// ---- GlobalTextList.TcGTLO
TEXTLIST GlobalTextList
  117 = ' MUST BE DISABLED'
  118 = ' MUST BE DISABLED TO RESUME'
  119 = ' MUST BE DISABLED TO RESUME NORMAL OPERATIONS'
  135 = ' MUST BE ENABLED FOR THRESHOLD AND FORCED CHECKS'
  134 = ' WILL PERFORM CHECK OPERATION ONCE AS NEXT TASK'
  33 = '%d'
  29 = '%i'
  55 = '%s'
  96 = '+1'
  126 = '+10'
  98 = '-1'
  127 = '-10'
  128 = '-50'
  4 = '1'
  5 = '2'
  70 = 'Auto Load'
  69 = 'Auto Unload'
  68 = 'AutoUnload'
  31 = 'Average Part Time'
  28 = 'Average Part Time: %d'
  165 = 'Backlash'
  64 = 'Batch'
  61 = 'Batch Process'
  170 = 'Box and Circle'
  24 = 'Clear Output'
  13 = 'Complete'
  35 = 'Completed'
  58 = 'Completed Part Count'
  18 = 'Completed Parts'
  41 = 'Completed Parts (Last 10)'
  75 = 'Completed Parts (newest first)'
  57 = 'CompletedPart Count'
  62 = 'Continual Process'
  1 = 'Create Part'
  111 = 'Diagnostics'
  110 = 'Enable / Disable'
  109 = 'Enable / Disable Position Check'
  121 = 'Enable / Disabling Position Checking'
  108 = 'Enable Position Check'
  122 = 'Enabling / Disabling Position Checking'
  164 = 'Encoder Slip'
  80 = 'End Effector'
  82 = 'End Effector 1'
  84 = 'End Effector Closed'
  86 = 'End Effector Grasp'
  83 = 'End Effector Open'
  85 = 'End Effector Part'
  107 = 'Error'
  157 = 'Fingers \nClosed'
  156 = 'Fingers \nOpen'
  90 = 'Fingers Closed'
  89 = 'Fingers Open'
  160 = 'Fixture'
  151 = 'Fofrces'
  154 = 'Force and Torqu Sensor'
  115 = 'Force Check'
  132 = 'Force Check Next'
  152 = 'Forces'
  136 = 'FT Sensor Controls'
  144 = 'Fx'
  143 = 'Fx (N)'
  145 = 'Fy'
  146 = 'Fz'
  159 = 'Grasped \nPart'
  158 = 'Grasped Part'
  155 = 'Gripper\nBody'
  91 = 'Gripper Body'
  21 = 'I1'
  92 = 'Induced Joint Error'
  99 = 'Induced Joint Error  (In 1/100 rad)'
  169 = 'Induced Robot Joint Error  (In 1/10 degrees)'
  105 = 'Induced Robot Joint Error  (In 1/100 rad)'
  39 = 'Input Position'
  3 = 'Insert Part'
  97 = 'J1'
  100 = 'J2'
  101 = 'J3'
  102 = 'J4'
  103 = 'J5'
  104 = 'J6'
  106 = 'Joint'
  23 = 'Load Input'
  166 = 'Mode'
  116 = 'MUST BE DISABLED'
  120 = 'MUST BE ENABLED FOR THRESHOLD AND FORCED CHECKS'
  147 = 'Newton-meter (N-m)'
  141 = 'Newtons'
  142 = 'Newtons (N)'
  171 = 'NIST Logo'
  22 = 'O1'
  163 = 'Off'
  63 = 'On Demand'
  131 = 'ONE TIME OPERATION'
  44 = 'Online Time'
  40 = 'Output Position'
  114 = 'Part Between Checks'
  124 = 'Part Between Checks Threshold'
  112 = 'Part Between Pos'
  32 = 'Part Count'
  30 = 'Part Count %i'
  27 = 'Part Count: %i'
  140 = 'Part Data Controls'
  8 = 'Part Fixture Time: '
  9 = 'Part Fixture Time: %s'
  88 = 'Part Grasped'
  59 = 'Part Number'
  15 = 'Part Removed'
  12 = 'Part Time: %d'
  11 = 'Part Time: %i'
  10 = 'Part Time: %s'
  36 = 'Part Type'
  113 = 'Parts Since Last Check'
  76 = 'Parts Since Pos Check'
  54 = 'Pick Frame'
  17 = 'Pick From WF'
  53 = 'Pick Location'
  60 = 'Place Frame'
  14 = 'Placed In WF'
  93 = 'Position Check'
  129 = 'Position Check Assigned Next'
  77 = 'Position Check Diagnostics'
  66 = 'Process Mode:\n%s'
  25 = 'Process Status:'
  26 = 'Process Status:\n%s'
  67 = 'Process Type:\n%s'
  51 = 'p_tas'
  2 = 'Remove Part'
  172 = 'Reserved'
  79 = 'Robot'
  78 = 'Robot Data Controls'
  130 = 'Sensor State'
  125 = 'Set at 50'
  123 = 'Settings'
  42 = 'Status'
  47 = 'Status\n%s'
  43 = 'Status: '
  137 = 'Switch FT Sensor Data Monitoring'
  138 = 'Switch FT Sensor Data Recording'
  139 = 'Switch Part Data Recording'
  65 = 'Switch Process Type'
  71 = 'Switch TCP/IP Data'
  72 = 'Switch TCP/IP Data Collection'
  74 = 'Switch TCP/IP Data Monitoring'
  73 = 'Switch TCP/IP Data Recording'
  94 = 'System Process'
  95 = 'System Settings'
  50 = 'Task'
  48 = 'Task Status\n%s'
  153 = 'Torques'
  34 = 'Trans'
  56 = 'Transfer'
  148 = 'Tx'
  149 = 'Ty'
  150 = 'Tz'
  19 = 'UR3'
  167 = 'UR3 Mode'
  46 = 'UR3 Power'
  45 = 'UR3 Status'
  173 = 'UR3 Task'
  20 = 'UR5'
  161 = 'UR5 Kinematic Chain'
  162 = 'UR5 Kinematic Chain Testing'
  168 = 'UR5 Mode'
  52 = 'UR5 Power'
  6 = 'WF1'
  7 = 'WF2'
  133 = 'WILL PERFORM CHECK OPERATION ONCE AS NEXT TASK'
  87 = 'Work Fix'
  16 = 'Work Fixture'
  81 = 'Work Fixtures'
  38 = 'Workfixture'
  37 = 'Workfixture Time (s)'
  0 = 'Workfixtures'
  49 = 'Workframe'
END_TEXTLIST

// ---- VISUs/ForceAndTorque.TcVIS
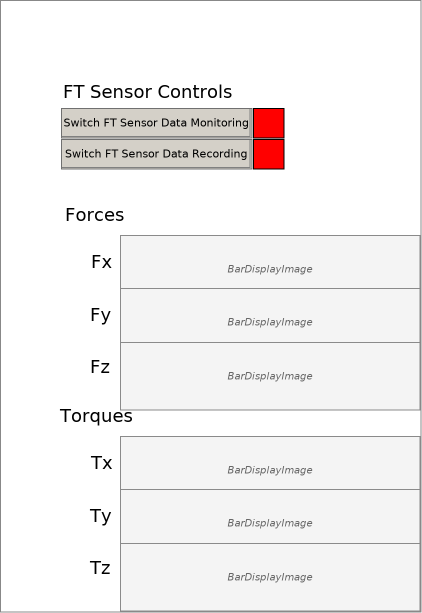
VISUALIZATION ForceAndTorque  // 422x613
    BarDisplayImage (120,235 300x68), value: Global.stFTData.Fx/10000, style: BarDisplayImage-Gray, scale format: %.1f, scale -5..5
        p518627256: Newtons (N)
    BarDisplayImage (120,288 300x68), value: Global.stFTData.Fy/10000, style: BarDisplayImage-Gray, scale format: %.1f, scale -5..5
        p518627256: Newtons (N)
    BarDisplayImage (120,342 300x68), value: Global.stFTData.Fz/10000, style: BarDisplayImage-Gray, scale format: %.1f, scale -5..5
        p518627256: Newtons (N)
    Label (88,247 34x30), "Fx"
    Label (87,300 34x30), "Fy"
    Label (87,352 34x30), "Fz"
    BarDisplayImage (120,436 300x68), value: Global.stFTData.Tx/100000, style: BarDisplayImage-Gray, scale format: %.1f, scale -1..1
        p518627256: Newton-meter (N-m)
    BarDisplayImage (120,489 300x68), value: Global.stFTData.Ty/100000, style: BarDisplayImage-Gray, scale format: %.1f, scale -1..1
        p518627256: Newton-meter (N-m)
    BarDisplayImage (120,543 300x68), value: Global.stFTData.Tz/100000, style: BarDisplayImage-Gray, scale format: %.1f, scale -1..1
        p518627256: Newton-meter (N-m)
    Label (88,448 34x30), "Tx"
    Label (87,501 34x30), "Ty"
    Label (87,553 34x30), "Tz"
    Label (62,197 98x36), "Forces"
    Label (57,398 98x36), "Torques"
    Button (61,108 191x30), "Switch FT Sensor Data Monitoring"
        OnMouseClick: toggle Global.bActivateFTDataCollection
    Button (61,139 191x30), "Switch FT Sensor Data Recording"
        OnMouseClick: toggle Global.bActivateFTDataRecording
    Rectangle (253,108 31x30), colour toggle: Global.bActivateFTDataCollection
    Rectangle (253,139 31x30), colour toggle: Global.bActivateFTDataRecording
    Label (60,77 246x30), "FT Sensor Controls"
END_VISUALIZATION

// ---- VISUs/PositionCheck.TcVIS
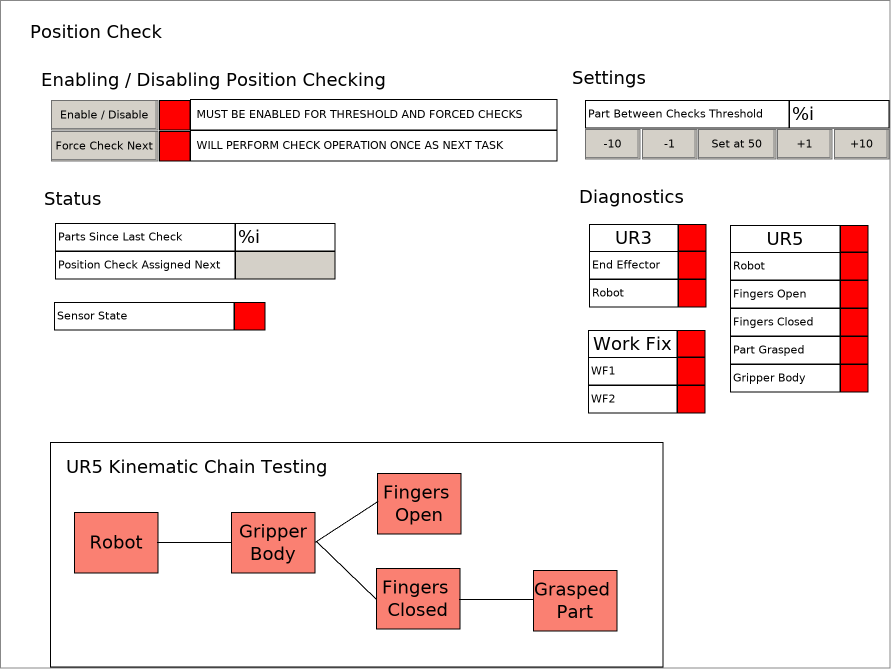
VISUALIZATION PositionCheck  // 891x669
    RoundedRectangle (50,442 613x225)
    Rectangle (55,223 180x28), "Parts Since Last Check"
    Rectangle (235,223 100x28), "%i", text variable: Global.nPartsSincePosCheck
    Rectangle (589,224 89x28), "UR3"
    Rectangle (589,251 89x28), "End Effector"
    Rectangle (589,279 89x28), "Robot"
    Rectangle (678,224 28x27), colour toggle: global.UR3PosCheck[1] and global.UR3PosCheck[2]
    Rectangle (678,279 28x28), colour toggle: Global.UR3PosCheck[2]
    Rectangle (678,251 28x28), colour toggle: Global.UR3PosCheck[1]
    Rectangle (730,225 110x28), "UR5"
    Rectangle (730,252 110x28), "Robot"
    Rectangle (730,280 110x28), "Fingers Open"
    Rectangle (840,225 28x27), colour toggle: Global.UR5PosCheck[1] and Global.UR5PosCheck[2] and Global.UR5PosCheck[3] and Global.UR5PosCheck[4] and Global.UR5PosCheck[5]
    Rectangle (840,280 28x28), colour toggle: Global.UR5PosCheck[3]
    Rectangle (840,252 28x28), colour toggle: Global.UR5PosCheck[5]
    Rectangle (588,330 89x28), "Work Fix"
    Rectangle (588,357 89x28), "WF1"
    Rectangle (588,385 89x28), "WF2"
    Rectangle (677,330 28x27)
    Rectangle (677,385 28x28)
    Rectangle (677,357 28x28)
    Rectangle (730,308 110x28), "Fingers Closed"
    Rectangle (840,308 28x28), colour toggle: Global.UR5PosCheck[2]
    Rectangle (730,336 110x28), "Part Grasped"
    Rectangle (840,336 28x28), colour toggle: Global.UR5PosCheck[1]
    Rectangle (730,364 110x28), "Gripper Body"
    Rectangle (840,364 28x28), colour toggle: Global.UR5PosCheck[4]
    Label (41,184 260x30), "Status"
    Button (51,100 107x30), "Enable / Disable"
        OnMouseClick: toggle Global.bEnablePosCheck
    Rectangle (159,100 31x30), colour toggle: Global.bEnablePosCheck
    Label (27,17 260x30), "Position Check"
    Rectangle (585,100 204x28), "Part Between Checks Threshold"
    Rectangle (789,100 100x28), "%i", text variable: Global.nPosCheckThreshold
    Button (51,131 107x30), "Force Check Next"
        OnMouseClick: toggle Global.bForcePosCheck
    Rectangle (159,131 31x30), colour toggle: Global.bForcePosCheck
    Rectangle (190,130 367x31), "WILL PERFORM CHECK OPERATION ONCE AS NEXT TASK"
    Rectangle (190,99 367x31), "MUST BE ENABLED FOR THRESHOLD AND FORCED CHECKS"
    Label (38,65 360x30), "Enabling / Disabling Position Checking"
    Label (569,63 260x30), "Settings"
    Button (698,129 78x30), "Set at 50"
        OnMouseClick: execute { Global.nPosCheckThreshold := 50; }
    Button (777,129 55x30), "+1"
        OnMouseClick: execute { Global.nPosCheckThreshold := Global.nPosCheckThreshold + 1; }
    Button (834,129 55x30), "+10"
        OnMouseClick: execute { Global.nPosCheckThreshold := Global.nPosCheckThreshold + 10; }
    Button (585,129 55x30), "-10"
        OnMouseClick: execute { Global.nPosCheckThreshold := Global.nPosCheckThreshold - 10; }
    Button (642,129 55x30), "-1"
        OnMouseClick: execute { Global.nPosCheckThreshold := Global.nPosCheckThreshold - 1; }
    Label (576,182 260x30), "Diagnostics"
    Rectangle (55,251 180x28), "Position Check Assigned Next"
    Rectangle (235,251 100x28), colour toggle: Global.bForcePosCheck
    Rectangle (54,302 180x28), "Sensor State"
    Rectangle (234,302 31x28), colour toggle: Global.bPosSensorState
    RoundedRectangle (74,512 84x61), "Robot", colour toggle: Global.UR5PosCheck[1]
    RoundedRectangle (231,512 84x61), "Gripper Body", colour toggle: Global.UR5PosCheck[2]
    RoundedRectangle (377,473 84x61), "Fingers Open", colour toggle: Global.UR5PosCheck[3]
    RoundedRectangle (376,568 84x61), "Fingers Closed", colour toggle: Global.UR5PosCheck[4]
    RoundedRectangle (533,570 84x61), "Grasped Part", colour toggle: Global.UR5PosCheck[5]
    Line (157,542) (231,542)
    Line (315,542) (378,501)
    Line (316,541) (376,599)
    Line (459,599) (533,599)
    Label (63,452 344x30), "UR5 Kinematic Chain Testing"
END_VISUALIZATION

// ---- VISUs/Settings.TcVIS
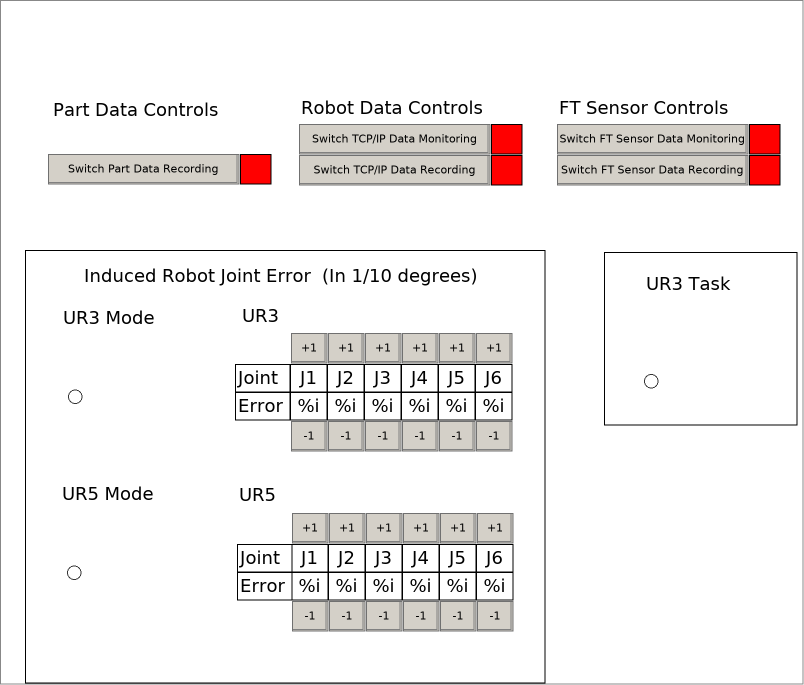
VISUALIZATION Settings  // 804x685
    RoundedRectangle (604,252 193x173)
    RoundedRectangle (25,250 520x433)
    Button (299,124 191x30), "Switch TCP/IP Data Monitoring"
        OnMouseClick: toggle Global.bActivateTCPIPDataCollection
    Button (299,155 191x30), "Switch TCP/IP Data Recording"
        OnMouseClick: toggle Global.bActivateTCPIPDataRecording
    Rectangle (491,124 31x30), colour toggle: Global.bActivateTCPIPDataCollection
    Rectangle (491,155 31x30), colour toggle: Global.bActivateTCPIPDataRecording
    Label (298,93 246x30), "Robot Data Controls"
    Label (81,261 507x30), "Induced Robot Joint Error (In 1/10 degrees)"
    Label (239,301 77x30), "UR3"
    Label (236,480 77x30), "UR5"
    Rectangle (291,572 37x28), "%i", text variable: Global.stUR5.InducedJointError[1]
    Button (292,513 36x30), "+1"
        OnMouseClick: execute { Global.stUR5.InducedJointError[1] := Global.stUR5.InducedJointError[1] + 1; }
    Button (292,601 36x30), "-1"
        OnMouseClick: execute { Global.stUR5.InducedJointError[1] := Global.stUR5.InducedJointError[1] - 1; }
    Rectangle (291,544 37x28), "J1"
    Rectangle (328,572 37x28), "%i", text variable: Global.stUR5.InducedJointError[2]
    Button (329,513 36x30), "+1"
        OnMouseClick: execute { Global.stUR5.InducedJointError[2] := Global.stUR5.InducedJointError[2] + 1; }
    Button (329,601 36x30), "-1"
        OnMouseClick: execute { Global.stUR5.InducedJointError[2] := Global.stUR5.InducedJointError[2] - 1; }
    Rectangle (328,544 37x28), "J2"
    Rectangle (365,572 37x28), "%i", text variable: Global.stUR5.InducedJointError[3]
    Button (366,513 36x30), "+1"
        OnMouseClick: execute { Global.stUR5.InducedJointError[3] := Global.stUR5.InducedJointError[3] + 1; }
    Button (366,601 36x30), "-1"
        OnMouseClick: execute { Global.stUR5.InducedJointError[3] := Global.stUR5.InducedJointError[3] - 1; }
    Rectangle (365,544 37x28), "J3"
    Rectangle (402,572 37x28), "%i", text variable: Global.stUR5.InducedJointError[4]
    Button (403,513 36x30), "+1"
        OnMouseClick: execute { Global.stUR5.InducedJointError[4] := Global.stUR5.InducedJointError[4] + 1; }
    Button (403,601 36x30), "-1"
        OnMouseClick: execute { Global.stUR5.InducedJointError[4] := Global.stUR5.InducedJointError[4] - 1; }
    Rectangle (402,544 37x28), "J4"
    Rectangle (439,572 37x28), "%i", text variable: Global.stUR5.InducedJointError[5]
    Button (440,513 36x30), "+1"
        OnMouseClick: execute { Global.stUR5.InducedJointError[5] := Global.stUR5.InducedJointError[5] + 1; }
    Button (440,601 36x30), "-1"
        OnMouseClick: execute { Global.stUR5.InducedJointError[5] := Global.stUR5.InducedJointError[5] - 1; }
    Rectangle (439,544 37x28), "J5"
    Rectangle (476,572 37x28), "%i", text variable: Global.stUR5.InducedJointError[6]
    Button (477,513 36x30), "+1"
        OnMouseClick: execute { Global.stUR5.InducedJointError[6] := Global.stUR5.InducedJointError[6] + 1; }
    Button (477,601 36x30), "-1"
        OnMouseClick: execute { Global.stUR5.InducedJointError[6] := Global.stUR5.InducedJointError[6] - 1; }
    Rectangle (476,544 37x28), "J6"
    Rectangle (237,544 55x28), "Joint"
    Rectangle (237,572 55x28), "Error", text variable: Global.stUR5.InducedJointError[1]
    Rectangle (290,392 37x28), "%i", text variable: Global.stUR3.InducedJointError[1]
    Button (291,333 36x30), "+1"
        OnMouseClick: execute { Global.stUR3.InducedJointError[1] := Global.stUR3.InducedJointError[1] + 1; }
    Button (291,421 36x30), "-1"
        OnMouseClick: execute { Global.stUR3.InducedJointError[1] := Global.stUR3.InducedJointError[1] - 1; }
    Rectangle (290,364 37x28), "J1"
    Rectangle (327,392 37x28), "%i", text variable: Global.stUR3.InducedJointError[2]
    Button (328,333 36x30), "+1"
        OnMouseClick: execute { Global.stUR3.InducedJointError[2] := Global.stUR3.InducedJointError[2] + 1; }
    Button (328,421 36x30), "-1"
        OnMouseClick: execute { Global.stUR3.InducedJointError[2] := Global.stUR3.InducedJointError[2] - 1; }
    Rectangle (327,364 37x28), "J2"
    Rectangle (364,392 37x28), "%i", text variable: Global.stUR3.InducedJointError[3]
    Button (365,333 36x30), "+1"
        OnMouseClick: execute { Global.stUR3.InducedJointError[3] := Global.stUR3.InducedJointError[3] + 1; }
    Button (365,421 36x30), "-1"
        OnMouseClick: execute { Global.stUR3.InducedJointError[3] := Global.stUR3.InducedJointError[3] - 1; }
    Rectangle (364,364 37x28), "J3"
    Rectangle (401,392 37x28), "%i", text variable: Global.stUR3.InducedJointError[4]
    Button (402,333 36x30), "+1"
        OnMouseClick: execute { Global.stUR3.InducedJointError[4] := Global.stUR3.InducedJointError[4] + 1; }
    Button (402,421 36x30), "-1"
        OnMouseClick: execute { Global.stUR3.InducedJointError[4] := Global.stUR3.InducedJointError[4] - 1; }
    Rectangle (401,364 37x28), "J4"
    Rectangle (438,392 37x28), "%i", text variable: Global.stUR3.InducedJointError[5]
    Button (439,333 36x30), "+1"
        OnMouseClick: execute { Global.stUR3.InducedJointError[5] := Global.stUR3.InducedJointError[5] + 1; }
    Button (439,421 36x30), "-1"
        OnMouseClick: execute { Global.stUR3.InducedJointError[5] := Global.stUR3.InducedJointError[5] - 1; }
    Rectangle (438,364 37x28), "J5"
    Rectangle (475,392 37x28), "%i", text variable: Global.stUR3.InducedJointError[6]
    Button (476,333 36x30), "+1"
        OnMouseClick: execute { Global.stUR3.InducedJointError[6] := Global.stUR3.InducedJointError[6] + 1; }
    Button (476,421 36x30), "-1"
        OnMouseClick: execute { Global.stUR3.InducedJointError[6] := Global.stUR3.InducedJointError[6] - 1; }
    Rectangle (475,364 37x28), "J6"
    Rectangle (235,364 55x28), "Joint"
    Rectangle (235,392 55x28), "Error", text variable: Global.stUR5.InducedJointError[1]
    Button (557,124 191x30), "Switch FT Sensor Data Monitoring"
        OnMouseClick: toggle Global.bActivateFTDataCollection
    Button (557,155 191x30), "Switch FT Sensor Data Recording"
        OnMouseClick: toggle Global.bActivateFTDataRecording
    Rectangle (749,124 31x30), colour toggle: Global.bActivateFTDataCollection
    Rectangle (749,155 31x30), colour toggle: Global.bActivateFTDataRecording
    Label (556,93 246x30), "FT Sensor Controls"
    Button (48,154 191x30), "Switch Part Data Recording"
        OnMouseClick: toggle Global.bActivatePartDataRecording
    Rectangle (240,154 31x30), colour toggle: Global.bActivatePartDataRecording
    Label (50,95 246x30), "Part Data Controls"
    RadioButton (66,350 150x93), variable: Global.stUR3.InducedJErrorType
        Areas[0]: Text=Off
        Areas[1]: Text=Encoder Slip
        Areas[2]: Text=Backlash
    Label (60,303 147x30), "UR3 Mode"
    RadioButton (65,526 150x93), variable: Global.stUR5.InducedJErrorType
        Areas[0]: Text=Off
        Areas[1]: Text=Encoder Slip
        Areas[2]: Text=Backlash
    Label (59,479 147x30), "UR5 Mode"
    RadioButton (642,306 150x150), variable: Global.nActiveUR3Task
        Areas[0]: Text=Box and Circle
        Areas[1]: Text=NIST Logo
        Areas[2]: Text=Reserved
    Label (643,269 103x30), "UR3 Task"
END_VISUALIZATION

// ---- VISUs/Process.TcVIS
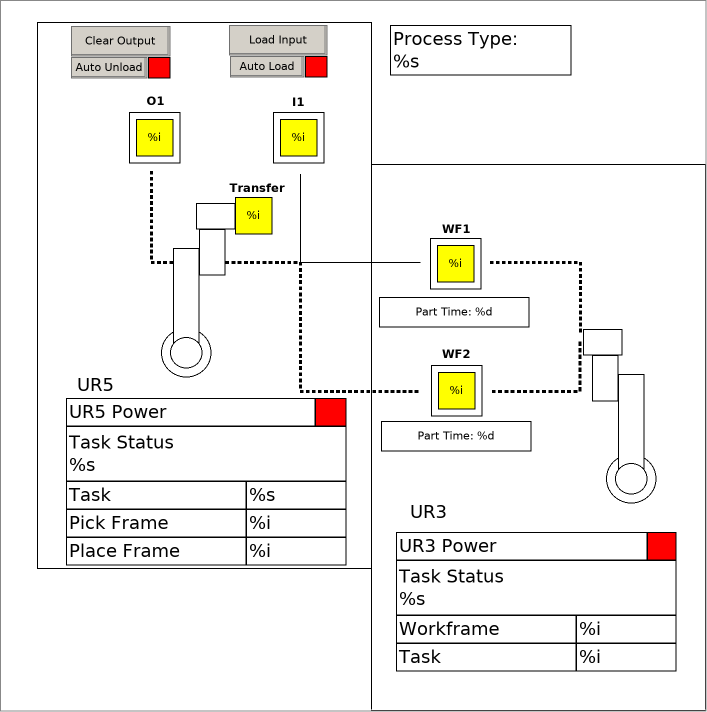
VISUALIZATION Process  // 707x712
    Rectangle (235,197 37x37)
    Line (371,164) (705,164)
    Line (371,710) (705,710)
    Line (705,164) (705,709)
    Line (371,164) (371,709)
    Rectangle (430,238 51x51), colour toggle: Global.arrWorkFixtures[1].bReserved
    Rectangle (431,365 51x51), colour toggle: Global.arrWorkFixtures[2].bReserved
    Rectangle (437,245 37x37), "%i", text variable: Global.arrWorkFixtures[1].stPart.nPartNumber, colour toggle: Global.arrWorkFixtures[1].stPart.bComplete, invisible if: NOT Global.arrWorkFixtures[1].stPart.bExists
    Rectangle (438,372 37x37), "%i", text variable: Global.arrWorkFixtures[2].stPart.nPartNumber, colour toggle: Global.arrWorkFixtures[2].stPart.bComplete, invisible if: NOT Global.arrWorkFixtures[2].stPart.bExists
    Rectangle (379,297 150x30), "Part Time: %d", text variable: Global.arrWorkFixtures[1].stPart.ntTimeInWorkfixture
    Rectangle (381,421 150x30), "Part Time: %d", text variable: Global.arrWorkFixtures[2].stPart.ntTimeInWorkfixture
    Line (37,22) (371,22)
    Line (37,568) (371,568)
    Line (371,22) (371,567)
    Line (37,23) (37,568)
    Label (67,370 57x30), "UR5"
    Rectangle (273,112 51x51), colour toggle: Global.arrInputFixtures[1].bReserved
    Rectangle (280,119 37x37), "%i", text variable: Global.arrInputFixtures[1].stPart.nPartNumber, colour toggle: Global.arrInputFixtures[1].stPart.bComplete, invisible if: NOT Global.arrInputFixtures[1].stPart.bExists
    Rectangle (129,112 51x51), colour toggle: Global.arrOutputFixtures[1].bReserved
    Rectangle (136,119 37x37), "%i", text variable: Global.arrOutputFixtures[1].stPart.nPartNumber, colour toggle: Global.arrOutputFixtures[1].stPart.bComplete, invisible if: NOT Global.arrOutputFixtures[1].stPart.bExists
    Button (229,25 98x30), "Load Input"
        OnMouseClick: execute { P_InputOutputHandling.bAddParts := TRUE; }
    Button (71,26 99x30), "Clear Output"
        OnMouseClick: execute { P_InputOutputHandling.bRemoveParts := true; }
    Line (300,262) (420,262), colour toggle: P_TaskHandling.stUR5TaskStatus.bInTask AND (P_TaskHandling.nUR5TargetPickFrame = Global.arrWorkFixtures[1].nWorkframe OR P_TaskHandling.nUR5TargetPlaceFrame = Global.arrWorkFixtures[1].nWorkframe)
    Line (300,174) (300,262), colour toggle: P_TaskHandling.nUR5TargetTask = 1
    Polyline (151,171) (151,262) (300,262), colour toggle: P_TaskHandling.nUR5TargetTask = 2
    Polyline (300,262) (300,391) (421,391), colour toggle: P_TaskHandling.stUR5TaskStatus.bInTask AND (P_TaskHandling.nUR5TargetPickFrame = Global.arrWorkFixtures[2].nWorkframe OR P_TaskHandling.nUR5TargetPlaceFrame = Global.arrWorkFixtures[2].nWorkframe)
    Rectangle (235,197 37x37), "%i", text variable: Global.stPartInTransit.nPartNumber, colour toggle: Global.stPartInTransit.bComplete, invisible if: NOT Global.stPartInTransit.bExists
    Polyline (490,262) (580,262) (580,335), colour toggle: P_TaskHandling.nUR3TargetWorkFixtureIndex = 1
    Polyline (492,391) (580,391) (580,339), colour toggle: P_TaskHandling.nUR3TargetWorkFixtureIndex = 2
    Rectangle (396,532 251x28), "UR3 Power"
    Rectangle (647,532 29x28), colour toggle: Global_Safety.UR3RedIND
    Rectangle (396,560 280x55), "Task Status %s", text variable: P_TaskHandling.stUR3TaskStatus.sRobotStatus
    Rectangle (396,615 180x28), "Workframe"
    Rectangle (576,615 100x28), "%i", text variable: P_TaskHandling.nUR3TargetWorkframe
    Rectangle (396,643 180x28), "Task"
    Rectangle (576,643 100x28), "%i", text variable: P_TaskHandling.nUR3TargetTask
    Rectangle (66,398 249x28), "UR5 Power"
    Rectangle (315,398 31x28), colour toggle: Global_Safety.UR5RedIND
    Rectangle (66,426 280x55), "Task Status %s", text variable: P_TaskHandling.stUR5TaskStatus.sRobotStatus
    Rectangle (66,481 180x28), "Task"
    Rectangle (246,481 100x28), "%s", text variable: P_TaskHandling.sUR5TargetTask
    Rectangle (66,509 180x28), "Pick Frame"
    Rectangle (246,509 100x28), "%i", text variable: P_TaskHandling.nUR5TargetPickFrame
    Label (400,497 57x30), "UR3"
    Rectangle (66,537 180x28), "Place Frame"
    Rectangle (246,537 100x28), "%i", text variable: P_TaskHandling.nUR5TargetPlaceFrame
    Group (161,203 74x174)
        Ellipse (0,125 50x49), colour toggle: Global_Safety.UR5RedIND
        Group (9,0 65x165)
            Rectangle (3,45 26x103)
            Rectangle (26,0 39x26)
            Ellipse (0,134 32x31)
            Rectangle (29,26 26x46)
    Group (583,329 73x174)
        Ellipse (23,125 50x49), colour toggle: Global_Safety.UR3RedIND
        Rectangle (35,45 26x103)
        Rectangle (0,0 39x26)
        Ellipse (32,134 32x31)
        Rectangle (9,26 26x46)
    Label (428,339 57x30), "WF2"
    Label (428,214 57x30), "WF1"
    Label (225,173 64x30), "Transfer"
    Label (270,87 57x30), "I1"
    Label (127,86 57x30), "O1"
    Rectangle (390,25 181x50), "Process Type: %s", text variable: P_InputOutputHandling.sProcessType
    Button (71,57 76x21), "Auto Unload"
        OnMouseClick: toggle P_InputOutputHandling.bAutoUnload
    Button (230,56 74x21), "Auto Load"
        OnMouseClick: toggle P_InputOutputHandling.bAutoLoad
    Rectangle (148,57 22x21), colour toggle: P_InputOutputHandling.bAutoUnload
    Rectangle (305,56 22x21), colour toggle: P_InputOutputHandling.bAutoLoad
END_VISUALIZATION

// ---- VISUs/TopVisu.TcVIS
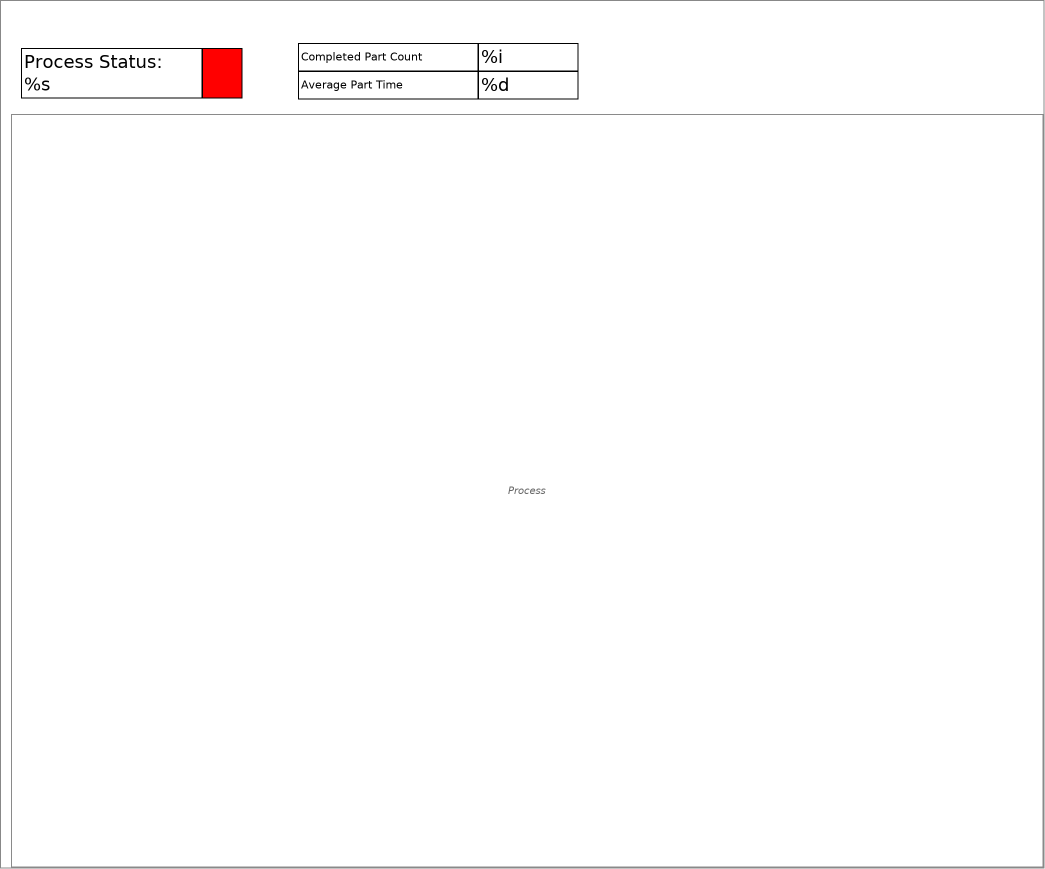
VISUALIZATION TopVisu  // 1045x869
    TabControl (11,114 1032x753)
        shows Process()
        shows PositionCheck()
        shows ForceAndTorque()
        shows Settings()
        [0]: TabTitle=System Process
        [1]: TabTitle=Position Check
        [2]: TabTitle=Force and Torqu Sensor
        [3]: TabTitle=System Settings
    Rectangle (202,48 40x50), colour toggle: MAIN.eProcessMode = E_ProcessModes.Running
    Rectangle (21,48 181x50), "Process Status: %s", text variable: MAIN.sProcessState
    Rectangle (298,43 180x28), "Completed Part Count"
    Rectangle (298,71 180x28), "Average Part Time"
    Rectangle (478,43 100x28), "%i", text variable: Global.nPartsCompleted
    Rectangle (478,71 100x28), "%d", text variable: Global.nAveragePartTime
END_VISUALIZATION
